Staubli VAL3: start.pgx

public program start()
begin
  call resetAllPallet()
end
